// Struckig
// Copyright (C) 2022 Stefan Besler

// This program is free software: you can redistribute it and/or modify
// it under the terms of the GNU General Public License as published by
// the Free Software Foundation, either version 3 of the License, or
// (at your option) any later version.

// This program is distributed in the hope that it will be useful,
// but WITHOUT ANY WARRANTY; without even the implied warranty of
// MERCHANTABILITY or FITNESS FOR A PARTICULAR PURPOSE.  See the
// GNU General Public License for more details.
//
// You should have received a copy of the GNU General Public License
// along with THIS PROGRAM.  IF NOT, see <http://www.gnu.org/licenses/>.
/// Checks whether a floating-point value is NaN.
/// Uses the IEEE-754 property that NaN is not equal to itself.
FUNCTION IsNaN : BOOL
VAR_INPUT
  value : LREAL; //< Input value.
END_VAR

IsNaN := value <> value;

END_FUNCTION

(* stored: Version 1.1.0.1
   POU IsNaN: Id {ea1d8573-8eaa-4d73-a977-92472b6d58b4}, SpecialFunc None *)
